ABB RobotStudio station: Project1.rsstnx

Station Project1 (saved by RobotStudio 24.3.10958.1)
Controller IRB120_3_58
  mechanical unit ROB_1: IRB120_3_58__01, 6 joints, base frame (0, 0, 0) mm
Layout (positions relative to the parent item):
  - IRB120_3_58__01 [mechanism, from %ABB.RobotStudio.Models.IRB120%\IRB120_3_58_G_01.rslib] at (0, 0, 0) mm; joint values [0, 0, -0.746, 0, 1.0662, 0] (rad or m)
  - Part_3 [part], size 200 x 200 x 200 mm
  - MyTool [mechanism, from Training Objects\myTool.rslib] at (242.63, 0, 793.7) mm, rotated rx 180 ry 71.65 rz 180 deg
  - Part_8 [part], size 398.6 x 396.9 x 396.9 mm
Attachment: MyTool is attached to IRB120_3_58__01 / Link6
Targets, tools, work objects and paths stored in the station, written as RAPID:
! task T_ROB1
MODULE CalibData
  PERS tooldata MyTool:=[TRUE,[[31.792631019,0,229.638935148],[0.945518576,0,0.325568154,0]],[1,[0,0,1],[1,0,0,0],0,0,0]];
ENDMODULE

